(* IEC 61131-3 sources: TcTidier/tests/fixtures/expected, 2 files *)

(* ---- interface_fixture.iecst ---- *)
FUNCTION InterfaceFixture : BOOL
VAR_INPUT
    enable : BOOL;
END_VAR
IF enable THEN
    InterfaceFixture := TRUE;
END_IF

(* ---- plain_text_fixture.st ---- *)
PROGRAM PlainTextFixture
VAR
    flag    : BOOL;
    counter : INT;
END_VAR
IF flag THEN
    counter := counter+1;
END_IF
